// TIA Portal V19 export
TYPE "type_errorInterface"
// stored: Access Published
   STRUCT
      parError : "type_parameterError";
   END_STRUCT;
END_TYPE
